Staubli VAL3: getSpeedDate.pgx

program getSpeedDate(string x_sSText, mdesc& x_mMdesc)
  local string l_sString[3]
  local bool l_bBool
  local num l_nNum
begin
  //获取速度参数
  call split(x_sSText,",",l_sString)
  //TXT文件会提供两个数值,前一个为加速度百分比，后一个为tvel
  //赋值
  //
  l_sString[0]=toNum(l_sString[0],x_mMdesc.accel,l_bBool)
  // x_mMdesc.decel=x_mMdesc.vel*x_mMdesc.accel
  x_mMdesc.decel=x_mMdesc.accel
  l_sString[1]=toNum(l_sString[1],x_mMdesc.tvel,l_bBool)


  //2015.02.04
  x_mMdesc.leave=0
  if l_sString[2]!=""
    toNum(l_sString[2],l_nNum,l_bBool)
    if l_bBool and l_nNum>0
      x_mMdesc.leave=l_nNum
    endIf
  endIf


end
